# EPICS substitutions: agpsApp/Db/system.substitutions
file system.template {
    pattern {SYS}
            {AGPS}
}
